// LS Electric XG5000 project: PLC_3
// PLC LSPLC
// module base 0 slot 0: Input/Output Module:XBC-DR30S (DC 24V Input 18 Contacts, Relay Output 12 Contacts)
// module base 0 slot 9: Analog Input Module:XBO-AD02A (A/D Voltage/Current Input Type(2 Channels))
// module base 0 slot 10: Analog Output Module:XBO-DA02A (D/A Voltage/Current Output Type(2 Channels))

PROGRAM NewProgram (task: Scan Program)

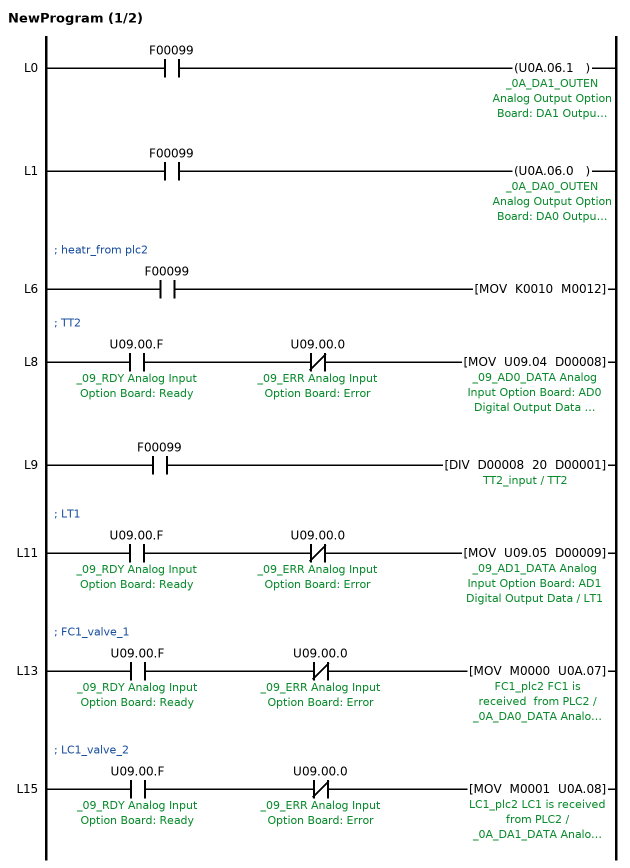
; L0
LOAD      F00099
OUT       U0A.06.1	// _0A_DA1_OUTEN Analog Output Option Board: DA1 Output Enable
; L1
LOAD      F00099
OUT       U0A.06.0	// _0A_DA0_OUTEN Analog Output Option Board: DA0 Output Enable
// heatr_from plc2
; L6
LOAD      F00099
MOV       K0010 M0012
// TT2
; L8
LOAD      U09.00.F	// _09_RDY Analog Input Option Board: Ready
AND NOT   U09.00.0	// _09_ERR Analog Input Option Board: Error
MOV       U09.04 D00008	// _09_AD0_DATA Analog Input Option Board: AD0 Digital Output Data / TT2_input
; L9
LOAD      F00099
DIV       D00008 20 D00001	// TT2_input / TT2
// LT1
; L11
LOAD      U09.00.F	// _09_RDY Analog Input Option Board: Ready
AND NOT   U09.00.0	// _09_ERR Analog Input Option Board: Error
MOV       U09.05 D00009	// _09_AD1_DATA Analog Input Option Board: AD1 Digital Output Data / LT1
// FC1_valve_1
; L13
LOAD      U09.00.F	// _09_RDY Analog Input Option Board: Ready
AND NOT   U09.00.0	// _09_ERR Analog Input Option Board: Error
MOV       M0000 U0A.07	// FC1_plc2 FC1 is received  from PLC2 / _0A_DA0_DATA Analog Output Option Board: DA0 Digital Input Data
// LC1_valve_2
; L15
LOAD      U09.00.F	// _09_RDY Analog Input Option Board: Ready
AND NOT   U09.00.0	// _09_ERR Analog Input Option Board: Error
MOV       M0001 U0A.08	// LC1_plc2 LC1 is received  from PLC2 / _0A_DA1_DATA Analog Output Option Board: DA1 Digital Input Data

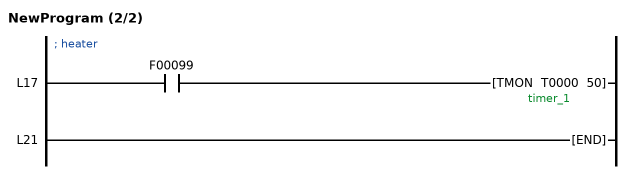
// heater
; L17
LOAD      F00099
TMON      T0000 50	// timer_1
; L21
END

VARIABLES AND COMMENTS (devices not used above)
P00040	BIT	heater
P00043	BIT	heater_lamp
K00000	BIT	J1
M0002	WORD	LC1_Virtual // LC1 is received from PLC 1 